// TwinCAT 3 PLC project _12_Composite
// ProgramVersion: 3.1.4023.0
// libraries:
//   Tc2_Standard, * (Beckhoff Automation GmbH)
//   Tc2_System, * (Beckhoff Automation GmbH)
//   Tc3_Module, * (Beckhoff Automation GmbH)
// project tree:
//   Composite Pattern/Abstraction/ Composite.TcPOU, E_Status.TcDUT, IComposite.TcIO
//   Composite Pattern/ Component.TcPOU, Machine.TcPOU, P_Composite.TcPOU, SubMachine1.TcPOU, SubMachine2.TcPOU
//   / MAIN.TcPOU, PlcTask.TcTTO
// (motion and I/O tree: see PLC project 13_decorator)
// real-time tasks:
//   TASK PlcTask: cycle T#10ms, priority 20, ADS port 350
// variable links:

CONFIGURATION _12_Composite
    RESOURCE PLC ON TwinCAT3
        TASK PlcTask(INTERVAL := T#10ms, PRIORITY := 20);
        PROGRAM MAIN WITH PlcTask : MAIN;
    END_RESOURCE
END_CONFIGURATION

// ---- Composite Pattern/Abstraction/E_Status.TcDUT
{attribute 'qualified_only'}
{attribute 'strict'}
{attribute 'to_string'}
TYPE E_Status :
(
	UNKNOWN := 0,
	IDLE,
	BUSY,
	DONE,
	ERROR := 666 
);
END_TYPE

// ---- Composite Pattern/Abstraction/IComposite.TcIO
INTERFACE IComposite

METHOD getChild : IComposite
VAR_INPUT
	child				: INT;
END_VAR
END_METHOD

METHOD getName : T_MAXSTRING
END_METHOD

METHOD getStatus : E_Status
VAR_INPUT
END_VAR
END_METHOD

METHOD logStatus
VAR_INPUT
END_VAR
END_METHOD

END_INTERFACE

// ---- MAIN.TcPOU
PROGRAM MAIN

(* 
	GOF 		Provide a unified interface to a set of interfaces in a subsystem. 
				Facade defines a higher-level interface that makes the subsystem easier to use.
*)
P_Composite();

END_PROGRAM

// ---- Composite Pattern/P_Composite.TcPOU
PROGRAM P_Composite
VAR
	machine01				: Machine;
END_VAR

machine01.logStatus();

END_PROGRAM

// ---- Composite Pattern/Machine.TcPOU
FUNCTION_BLOCK Machine EXTENDS Composite
VAR
	subMachine01				: SubMachine1;
	subMachine02				: SubMachine2;	
	childs						: ARRAY[1..NOOFCHILDS] OF IComposite := [subMachine01,subMachine02]; 	
END_VAR
VAR CONSTANT
	NOOFCHILDS					: INT := 2;
END_VAR

METHOD logStatus
VAR
	sMessage				: STRING;		
	i						: DINT;
END_VAR
// Local status 
SUPER^.logStatus();

// Loop through childs
FOR i := 1 TO NOOFCHILDS DO
	IF childs[i]<>0 THEN
		childs[i].logStatus();
	END_IF
END_FOR
END_METHOD

END_FUNCTION_BLOCK

// ---- Composite Pattern/Abstraction/Composite.TcPOU
{attribute 'reflection'}
FUNCTION_BLOCK ABSTRACT Composite IMPLEMENTS IComposite
VAR
	{attribute 'instance-path'}
	{attribute 'noinit'}
	instancePath			: STRING;	
	
	// Local status
	_status					: E_Status;	
	_statusPrev				: E_Status := 666; 
END_VAR

METHOD getChild : IComposite
VAR_INPUT
	child	: INT;
END_VAR
// default implementation, return empty
getChild := 0;
END_METHOD

METHOD getName : Tc2_System.T_MaxString
// default implementation, return empty string
getName := instancePath;
END_METHOD

METHOD getStatus : E_Status
// default implementation, return status unknown
getStatus := _status;
END_METHOD

METHOD logStatus
VAR
	sMessage				: STRING;		
END_VAR
// default implementation, do nothing
IF (_statusPrev <> _status)	THEN
	sMessage := concat(concat(instancePath, ': '), TO_STRING(_status));
	adsLogStr(	msgCtrlMask		:= ADSLOG_MSGTYPE_LOG,
			msgFmtStr 		:= '%s',
			strArg			:= sMessage 
			);	
	_statusPrev := _status;
END_IF
END_METHOD

END_FUNCTION_BLOCK

// ---- Composite Pattern/SubMachine1.TcPOU
FUNCTION_BLOCK SubMachine1 extends Composite
VAR
	component1					: Component;
	component2					: Component;
	childs						: ARRAY[1..NOOFCHILDS] OF IComposite := [component1,component2]; 
END_VAR
VAR CONSTANT
	NOOFCHILDS					: INT := 2;
END_VAR

METHOD logStatus
VAR
	sMessage				: STRING;		
	i						: DINT;
END_VAR
// Local status 
SUPER^.logStatus();

// Loop through childs
FOR i := 1 TO NOOFCHILDS DO
	IF childs[i]<>0 THEN
		childs[i].logStatus();
	END_IF
END_FOR
END_METHOD

END_FUNCTION_BLOCK

// ---- Composite Pattern/Component.TcPOU
FUNCTION_BLOCK Component EXTENDS Composite
VAR
END_VAR

METHOD logStatus
VAR
	sMessage				: STRING;		
END_VAR
// Local status 
SUPER^.logStatus();
END_METHOD

END_FUNCTION_BLOCK

// ---- Composite Pattern/SubMachine2.TcPOU
FUNCTION_BLOCK SubMachine2 extends Composite
VAR
	component1					: Component;
	component2					: Component;
	component3					: Component;
	childs						: ARRAY[1..NOOFCHILDS] OF IComposite := [component1,component2,component3]; 	
END_VAR
VAR CONSTANT
	NOOFCHILDS					: INT := 3;
END_VAR

METHOD logStatus
VAR
	sMessage				: STRING;		
	i						: DINT;
END_VAR
// Local status 
SUPER^.logStatus();

// Loop through childs
FOR i := 1 TO NOOFCHILDS DO
	IF childs[i]<>0 THEN
		childs[i].logStatus();
	END_IF
END_FOR
END_METHOD

END_FUNCTION_BLOCK
